// TwinCAT 3 PLC project pruebaPickAndPlace
// ProgramVersion: 3.1.4024.0
// libraries:
//   Tc2_Standard, * (Beckhoff Automation GmbH)
//   Tc2_System, * (Beckhoff Automation GmbH)
//   Tc3_Module, * (Beckhoff Automation GmbH)
//   VisuSymbols,3.5.10.0,System
// project tree:
//   / GlobalTextList.TcGTLO, PlcTask.TcTTO, Visualization Manager.TcVMO (not stored)
//   GVLs/ GVLvars.TcGVL
//   POUs/ MAIN.TcPOU
//   VISUs/ HMI.TcVIS
// real-time tasks:
//   TASK PlcTask: cycle T#10ms, priority 20, ADS port 350

CONFIGURATION pruebaPickAndPlace
    RESOURCE PLC ON TwinCAT3
        TASK PlcTask(INTERVAL := T#10ms, PRIORITY := 20);
        PROGRAM MAIN WITH PlcTask : MAIN;
    END_RESOURCE
END_CONFIGURATION

// ---- GVLs/GVLvars.TcGVL
{attribute 'qualified_only'}
VAR_GLOBAL
	
	// Barra Posicionamiento Bases
	{attribute 'OPC.UA.DA' := '1'}
	cerrarAbrazaderaBase : BOOL;
	{attribute 'OPC.UA.DA' := '1'}
	levantarAbrazaderaBase : BOOL;
	{attribute 'OPC.UA.DA' := '1'}
	limiteSujeccionBase : BOOL;
	{attribute 'OPC.UA.DA' := '1'}
	limiteVerticalBase : BOOL;
	
	// Barra posicionamiento Tapas
 	{attribute 'OPC.UA.DA' := '1'}
	levantarAbrazaderaTapa : BOOL;
	{attribute 'OPC.UA.DA' := '1'}
	cerrarAbrazaderaTapa : BOOL;
	{attribute 'OPC.UA.DA' := '1'}
	limiteSujeccionTapa : BOOL;
	{attribute 'OPC.UA.DA' := '1'}
	limiteVerticalTapa : BOOL;
 
	// SENSORES
	{attribute 'OPC.UA.DA' := '1'}
	sensorFotoBase : BOOL;;
	{attribute 'OPC.UA.DA' := '1'}
	sensorFotoTapa : BOOL;
	{attribute 'OPC.UA.DA' := '1'}
	sensorPostSellado : BOOL;
	{attribute 'OPC.UA.DA' := '1'}
	modoManual : BOOL; // Estado 0 del selector
	{attribute 'OPC.UA.DA' := '1'}
	modoAuto : BOOL; // Estado 1 del selector

	
	// Pick & Place

	{attribute 'OPC.UA.DA' := '1'}
	PickPlace_MoverX : BOOL;
	{attribute 'OPC.UA.DA' := '1'}
	PickPlace_MoverZ : BOOL;
	{attribute 'OPC.UA.DA' := '1'}
	PickPlace_Agarrar : BOOL;
	{attribute 'OPC.UA.DA' := '1'}
	PickPlace_Detectado : BOOL;
	{attribute 'OPC.UA.DA' := '1'}
	PickPlace_MovingXY: BOOL;
	{attribute 'OPC.UA.DA' := '1'}
	PickPlace_MovingZ: bool; 
	
	
	// CINTAS
	{attribute 'OPC.UA.DA' := '1'}
	cintaBases : BOOL;
	{attribute 'OPC.UA.DA' := '1'}
	cintaTapas : BOOL;
	
	// CUADRO
	{attribute 'OPC.UA.DA' := '1'}
	 botonStart : BOOL;
	{attribute 'OPC.UA.DA' := '1'}
	 botonStop : BOOL;	
	 {attribute 'OPC.UA.DA' := '1'}
	 botonReset : BOOL;
	{attribute 'OPC.UA.DA' := '1'}
	 luzVerticalVerde : BOOL;
	{attribute 'OPC.UA.DA' := '1'}
	 luzVerticalNaranja : BOOL;
	{attribute 'OPC.UA.DA' := '1'}
	 luzVerticalRoja : BOOL;	
	{attribute 'OPC.UA.DA' := '1'}
	 luzStop : BOOL;  // luz de boton stop
	 {attribute 'OPC.UA.DA' := '1'}
	 luzStart : BOOL; // luz del boton de start
	 {attribute 'OPC.UA.DA' := '1'}
	 luzReset : BOOL; 
	 {attribute 'OPC.UA.DA' := '1'}
	 seta : BOOL; // Seta de emergencia
 

 
END_VAR

// ---- POUs/MAIN.TcPOU
PROGRAM MAIN
VAR
	sistemaActivo : BOOL;
	
	cintaBase : BOOL;
	cintaTapa : BOOL;
	
	
	baseOK: BOOL;
	tapaOK: BOOL;
	flancoBajada_MovingXY: BOOL;
	movingXY_Anterior: BOOL;
	flancoBajada_MovingZ: BOOL;
	movingZ_Anterior: BOOL;
	EstadoPickPlace: INT;
	timerMovimiento: TON;
	tiempoMovimiento: TIME;
	
	flancoTapa : F_TRIG;
	flancoBase : F_TRIG;
	luzVerde: BOOL;
	luzNaranja: BOOL;
	luzRojo: BOOL;
	luzStop: BOOL;
	luzStart: BOOL;
	luzReset: BOOL;
	emergencia: BOOL;
	ProductoFinal: BOOL;
END_VAR

luzStop := FALSE;
luzStart := FALSE;
luzReset := FALSE;

//Si se pulsa el boton de start se arrancan als cintas
IF GVLvars.botonStart AND NOT emergencia THEN
	sistemaActivo := TRUE;
	luzVerde := TRUE;
	luzNaranja := FALSE;
	luzRojo := FALSE;
	luzStop := FALSE;
	luzStart := TRUE;
	
END_IF

IF NOT GVLvars.botonStop AND NOT emergencia THEN
	luzReset := TRUE;
	sistemaActivo := FALSE;
	cintaBase := FALSE;
	cintaTapa := FALSE;
	luzVerde := FALSE;
	luzNaranja := TRUE;
	luzRojo := FALSE;
	
END_IF


IF NOT GVLvars.seta THEN
	sistemaActivo := FALSE;
	cintaBase := FALSE;
	cintaTapa := FALSE;
	luzVerde := FALSE;
	luzNaranja := FALSE;
	luzRojo := TRUE;
	emergencia := TRUE;
END_IF


IF  GVLvars.seta AND emergencia THEN
	IF GVLvars.botonReset THEN
		sistemaActivo := TRUE;
		luzVerde := TRUE;
		luzNaranja := FALSE;
		luzRojo := FALSE;
		luzStop := FALSE;
		luzStart := FALSE;
		luzReset := TRUE;
		emergencia := FALSE;
	END_IF
END_IF

IF sistemaActivo AND emergencia = FALSE THEN
	
	IF baseOK = FALSE AND tapaOK = FALSE THEN
		cintaBase := TRUE;
	cintaTapa := TRUE;
	END_IF
	
	flancoTapa(CLK:=GVLvars.sensorFotoTapa);
	flancoBase(CLK:= GVLvars.sensorFotoBase);
	
	// Base en barrera posicionadora
	IF  flancoBase.Q THEN
		baseOK := TRUE;
		cintaBase := FALSE;
		
		GVLvars.cerrarAbrazaderaBase := TRUE;
	END_IF
	
	// Tapa en barrera posiconadora
	IF flancoTapa.Q THEN
		tapaOK := TRUE;
		cintaTapa := FALSE;
		GVLvars.cerrarAbrazaderaTapa := TRUE;
	END_IF
	
//	// --- Detección de flancos ---
//	flancoBajada_MovingXY := (NOT GVL_Var.PickPlace_MovingXY) AND movingXY_Anterior;
//	flancoBajada_MovingZ := (NOT GVL_Var.PickPlace_MovingZ) AND movingZ_Anterior;
	
//	movingXY_Anterior := GVL_Var.PickPlace_MovingXY;
//	movingZ_Anterior := GVL_Var.PickPlace_MovingZ;
	
	// --- Maquina de estados Pick & Place ---
	CASE EstadoPickPlace OF
	
		0: 
			
			// Inicio - piezas posicionadas y abrazaderas cerradas
			IF baseOK AND tapaOK AND GVLvars.limiteSujeccionBase AND GVLvars.limiteSujeccionTapa THEN
				EstadoPickPlace := 1;
			END_IF
	
		1: // Desplagar horizontalmente
			GVLvars.PickPlace_MoverZ := FALSE; // vertical
			GVLvars.PickPlace_MoverX := TRUE; //  horizontal
			GVLvars.PickPlace_Agarrar := FALSE; // ventosa
			ProductoFinal := FALSE;

			// EBERIA SER CON FLANCOS
			// si esta comletamnte extentida horizontalmente -> siguiente estao
			IF NOT GVLvars.PickPlace_MovingXY THEN
				timerMovimiento(IN:=TRUE, PT:=T#2S);
				IF timerMovimiento.Q THEN
//				GVL_Var.PickPlace_MoverZ := FALSE;
				timerMovimiento(IN:=FALSE);
	
				EstadoPickPlace := 2;
			END_IF
				
			END_IF
	
		2: // Bajamos vertical
			GVLvars.PickPlace_MoverZ := TRUE; //desplargar vertical
			GVLvars.PickPlace_MoverX := TRUE; // esplagamos horizontal
			GVLvars.PickPlace_Agarrar := FALSE; // ventosa

			// DEBERIA SER CON FLANCOS
			// si esta comletamnte extentida horizontalmente -> siguiente estao
			IF NOT GVLvars.PickPlace_MovingZ THEN
				EstadoPickPlace := 3;
			END_IF
	
		3: // AGARRAR objeto
			GVLvars.PickPlace_MoverZ := TRUE;  
			GVLvars.PickPlace_MoverX := TRUE;
			GVLvars.PickPlace_Agarrar := TRUE;
	
			
			timerMovimiento(IN:=TRUE, PT:=T#2S);
			IF timerMovimiento.Q THEN
//				GVL_Var.PickPlace_MoverZ := FALSE;
				timerMovimiento(IN:=FALSE);
	
				EstadoPickPlace := 4;
			END_IF
	
		4: // recogemos verticalmente ocn objeto agarrado
			GVLvars.PickPlace_MoverZ := FALSE;  
			GVLvars.PickPlace_MoverX := TRUE;
			GVLvars.PickPlace_Agarrar := TRUE;
	

			// DEBERIA SER CON FLANCOS
			// si esta comletamnte extentida horizontalmente -> siguiente estao
			IF NOT GVLvars.PickPlace_MovingZ THEN
				
			timerMovimiento(IN:=TRUE, PT:=T#2S);
			IF timerMovimiento.Q THEN
//				GVL_Var.PickPlace_MoverZ := FALSE;
				timerMovimiento(IN:=FALSE);
	
				EstadoPickPlace := 5;
			END_IF
				
			END_IF
	
		5: // recogemos horizontal con pieza aujeta
			GVLvars.PickPlace_MoverZ := FALSE;  
			GVLvars.PickPlace_MoverX := FALSE;
			GVLvars.PickPlace_Agarrar := TRUE;
			
			//GVL_Var.cerrarAbrazaderaBase := FALSE;
	

			IF NOT GVLvars.PickPlace_MovingXY THEN
				
			timerMovimiento(IN:=TRUE, PT:=T#2S);
			IF timerMovimiento.Q THEN
//				GVL_Var.PickPlace_MoverZ := FALSE;
				timerMovimiento(IN:=FALSE);
				EstadoPickPlace := 6;
				
			END_IF
					
			END_IF
	
		6: //bajar verticalmente
			GVLvars.PickPlace_MoverZ := TRUE;  
			GVLvars.PickPlace_MoverX := FALSE;
			GVLvars.PickPlace_Agarrar := TRUE;
	
		
			IF NOT GVLvars.PickPlace_MovingZ THEN
				
			timerMovimiento(IN:=TRUE, PT:=T#2S);
			IF timerMovimiento.Q THEN
//				GVL_Var.PickPlace_MoverZ := FALSE;
				timerMovimiento(IN:=FALSE);
	
				EstadoPickPlace := 7;
			END_IF
			END_IF
							


	
		7: // soltar objeto
			GVLvars.PickPlace_MoverZ := TRUE;  
			GVLvars.PickPlace_MoverX := FALSE;
			GVLvars.PickPlace_Agarrar := FALSE;
	
			// Reiniciar variables y continuar producción
			estadoPickPlace := 8;
			
			
		8:
			GVLvars.PickPlace_MoverZ := FALSE;  
			GVLvars.PickPlace_MoverX := FALSE;
			GVLvars.PickPlace_Agarrar := FALSE;
			
			IF NOT GVLvars.PickPlace_MovingZ THEN		
					EstadoPickPlace := 9;
			END_IF
			
		//Estado para levantar a barreara de posicionameinto
		// e arranque de cintas
		9:
			GVLvars.levantarAbrazaderaTapa := TRUE;
			cintaBase := TRUE;
			cintaTapa := TRUE;
			ProductoFinal := TRUE;
			
			//Si lla paso la barrera posicionadora
			IF GVLvars.sensorPostSellado THEN
				GVLvars.levantarAbrazaderaTapa := FALSE;
				baseOK := FALSE;
				tapaOK := FALSE;
	
				GVLvars.cerrarAbrazaderaBase := FALSE;
				GVLvars.cerrarAbrazaderaTapa := FALSE;
	
				EstadoPickPlace := 0;
			END_IF
	
	ELSE
		EstadoPickPlace := 0; // Si estado inválido, reiniciar
	END_CASE	
END_IF

// Se actualizan las salias
GVLvars.cintaBases := cintaBase;
GVLvars.cintaTapas := cintaTapa;
GVLvars.luzVerticalNaranja := luzNaranja;
GVLvars.luzVerticalRoja := luzRojo;
GVLvars.luzVerticalVerde := luzVerde;
GVLvars.luzStop := luzStop;
GVLvars.luzStart := luzStart;
GVLvars.luzReset := luzReset;
//GVL_Var.cerrarAbrazaderaBase :=
//GVL_Var.cerrarAbrazaderaTapa
//GVL_Var.levantarAbrazaderaBase
//GVL_Var.levantarAbrazaderaTapa
//GVL_Var.PickPlace_Agarrar
//GVL_Var.PickPlace_MoverX
//GVL_Var.PickPlace_MoverZ

END_PROGRAM

// ---- GlobalTextList.TcGTLO
TEXTLIST GlobalTextList
  30 = 'Abrazadera Base'
  360 = 'Abrazadera Tapa'
  436 = 'Cinta con Bases'
  679 = 'Cinta con las bases y posteriormente producto final'
  348 = 'Cinta con las tapas '
  583 = 'Cinta con Tapas'
  357 = 'Desplegando Brazo Horizontal '
  94 = 'Desplegando Brazo X'
  193 = 'Desplegando Brazo Z'
  646 = 'Detección de objeto'
  41 = 'Detección del objeto por parte del Pick&Place'
  305 = 'mover Brazo Z'
  275 = 'Producto Listo '
  341 = 'Recogiendo Brazo Horizontal '
  51 = 'Recogiendo Brazo Z'
  389 = 'Reset'
  857 = 'Seta'
  747 = 'Start'
  828 = 'Stop'
  394 = 'Sujeccion de Tapa (Ventosa)'
END_TEXTLIST

// ---- VISUs/HMI.TcVIS
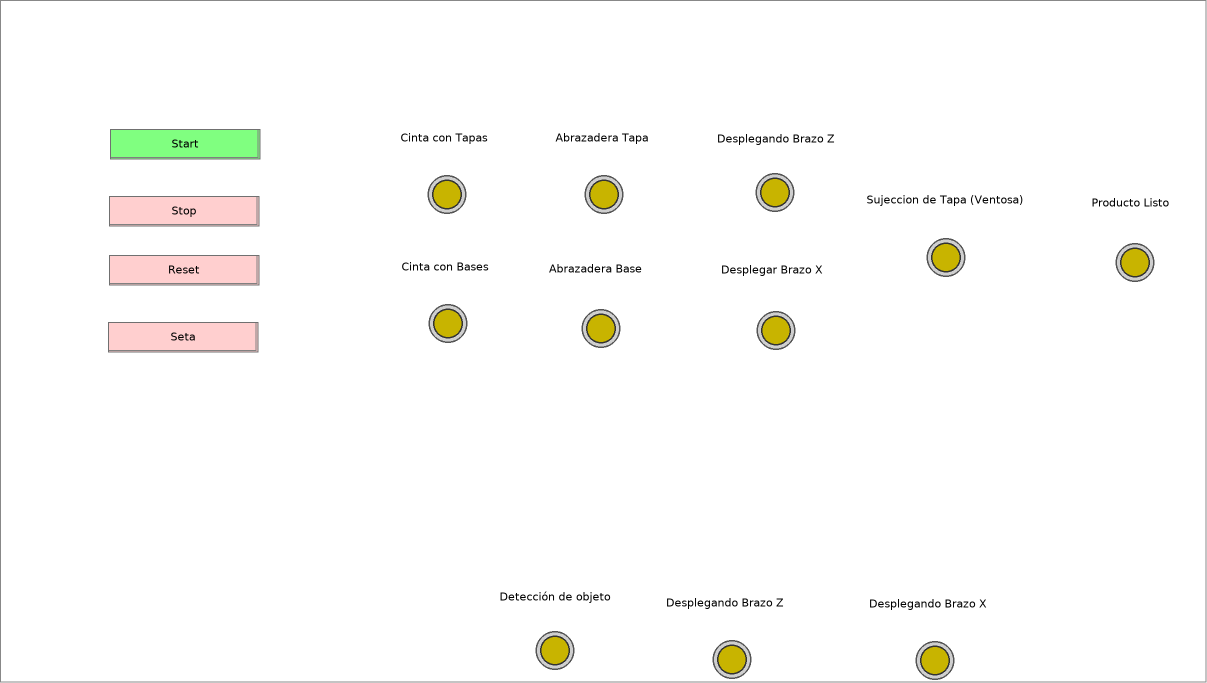
VISUALIZATION HMI  // 1207x683
    Button (110,129 150x30), "Start"
        toggle GVLvars.botonStart
    Button (109,196 150x30), "Stop"
        toggle GVLvars.botonStop
    Button (109,255 150x30), "Reset"
        toggle GVLvars.botonReset
    Button (108,322 150x30), "Seta"
        toggle GVLvars.seta
    Lamp1 (1109,240 52x45), variable: MAIN.ProductoFinal, style: Lamp-Lamp1-Yellow
    Label (1057,188 150x30), "Producto Listo"
    Lamp1 (421,172 52x45), tooltip "Cinta con las bases y posteriormente producto final", variable: GVLvars.cintaBases, style: Lamp-Lamp1-Yellow
    Label (369,123 150x30), "Cinta con Tapas"
    Lamp1 (422,301 52x45), tooltip "Cinta con las tapas", variable: GVLvars.cintaTapas, style: Lamp-Lamp1-Yellow
    Label (370,252 150x30), "Cinta con Bases"
    Lamp1 (706,637 52x45), tooltip "Cinta con las bases y posteriormente producto final", variable: GVLvars.PickPlace_MovingZ, style: Lamp-Lamp1-Yellow
    Label (630,582 190x42), "Desplegando Brazo Z"
    Lamp1 (749,170 52x45), tooltip "Cinta con las bases y posteriormente producto final", variable: GVLvars.PickPlace_MoverZ, style: Lamp-Lamp1-Yellow
    Label (681,118 190x42), "Desplegando Brazo Z"
    Lamp1 (909,638 52x45), tooltip "Cinta con las bases y posteriormente producto final", variable: GVLvars.PickPlace_MovingXY, style: Lamp-Lamp1-Yellow
    Label (833,583 190x42), "Desplegando Brazo X"
    Lamp1 (750,308 52x45), tooltip "Cinta con las bases y posteriormente producto final", variable: GVLvars.PickPlace_MoverX, style: Lamp-Lamp1-Yellow
    Label (677,249 190x42), "Desplegar Brazo X"
    Lamp1 (920,235 52x45), variable: GVLvars.PickPlace_Agarrar, style: Lamp-Lamp1-Yellow
    Label (849,185 192x30), "Sujeccion de Tapa (Ventosa)"
    Lamp1 (578,172 52x45), tooltip "Cinta con las bases y posteriormente producto final", variable: GVLvars.cerrarAbrazaderaTapa, style: Lamp-Lamp1-Yellow
    Label (548,117 108x42), "Abrazadera Tapa"
    Lamp1 (575,306 52x45), tooltip "Cinta con las bases y posteriormente producto final", variable: GVLvars.cerrarAbrazaderaBase, style: Lamp-Lamp1-Yellow
    Label (538,248 115x42), "Abrazadera Base"
    Lamp1 (529,628 52x45), tooltip "Detección del objeto por parte del Pick&Place", variable: GVLvars.PickPlace_Detectado, style: Lamp-Lamp1-Yellow
    Label (459,582 192x30), "Detección de objeto"
END_VISUALIZATION
